FUNCTION_BLOCK FB_MotionAxisNCOld IMPLEMENTS I_MotionAxisOld
VAR
    iHome : I_Home;
    iHalt : I_Halt;
    iPower : I_Power;
    iReset : I_Reset;
    iMoveAbsolute : I_MoveAbsolute;
    iReadParameter : I_ReadParameter;
    iWriteParameter  : I_WriteParameter;
    iParamSaveRestore: I_ParamSaveRestore;
    iEncoderScaling : I_EncoderScaling;
    iAxisStatus : I_AxisStatus;
    iBacklashCompensation : I_BacklashCompensation;
    bError: BOOL;
    nErrorID: UDINT;
    sMessage : T_MAXSTRING;
    rtAbortDone : R_TRIG;

END_VAR

(*
    Error from NC functions
    The error will be sent to EPICS interface based on predifined
    priority: axis, power, backlash, absoluteMove, etc...
*)
IF THIS^.iPower.Error AND THIS^.iPower.PowerIsEnabled THEN
    bError:=THIS^.iPower.Error;
    nErrorId:=THIS^.iPower.ErrorID;
    sMessage := THIS^.iPower.Message;
ELSIF THIS^.iHalt.Error AND THIS^.iHalt.Active THEN
    bError:=THIS^.iHalt.Error;
    nErrorId:=THIS^.iHalt.ErrorID;
    sMessage := THIS^.iHalt.Message;
ELSIF THIS^.iReset.Error AND THIS^.iReset.Active THEN
    bError:=THIS^.iReset.Error;
    nErrorId:=THIS^.iReset.ErrorID;
    sMessage := THIS^.iReset.Message;
ELSIF THIS^.iBacklashCompensation.Error THEN
    bError:=THIS^.iBacklashCompensation.Error;
    nErrorId:=THIS^.iBacklashCompensation.ErrorID;
    sMessage := THIS^.iBacklashCompensation.Message;
ELSIF THIS^.iMoveAbsolute.Error THEN
    bError:=THIS^.iMoveAbsolute.Error;
    nErrorId:=THIS^.iMoveAbsolute.ErrorID;
    sMessage := THIS^.iMoveAbsolute.Message;
ELSIF THIS^.iHome.Error (*Homing error*) THEN
    bError:=THIS^.iHome.Error;
    nErrorId:=THIS^.iHome.ErrorID;
    sMessage := THIS^.iHome.Message;
ELSIF THIS^.iAxisStatus.Error  THEN
    bError:=THIS^.iAxisStatus.Error;
    nErrorId:=THIS^.iAxisStatus.ErrorID;
    sMessage := THIS^.iAxisStatus.Message;
ELSIF THIS^.iReadParameter.Error THEN
    bError := THIS^.iReadParameter.Error;
    nErrorId := THIS^.iReadParameter.ErrorID;
    sMessage := THIS^.iReadParameter.Message;
ELSIF THIS^.iWriteParameter.Error THEN
    bError := THIS^.iWriteParameter.Error;
    nErrorId := THIS^.iWriteParameter.ErrorID;
    sMessage := THIS^.iWriteParameter.Message;
ELSIF THIS^.iParamSaveRestore.Error THEN
    bError := THIS^.iParamSaveRestore.Error;
    nErrorId := THIS^.iParamSaveRestore.ErrorID;
    sMessage := THIS^.iParamSaveRestore.Message;
ELSE
    bError:=FALSE;
    nErrorId:=0;
    sMessage := '';
END_IF;

PROPERTY AbortDone : BOOL
GET
AbortDone := THIS^.iHalt.Done OR THIS^.iReset.Done;
END_GET
END_PROPERTY

PROPERTY Aborted : BOOL
GET
ABorted := THIS^.iMoveAbsolute.Aborted;
END_GET
END_PROPERTY

METHOD AxisEnabled : BOOL
VAR_INPUT
END_VAR
AxisEnabled:=THIS^.iAxisStatus.AxisEnabled();
END_METHOD

PROPERTY AxisReadParamsInit : BOOL
GET
AxisReadParamsInit := THIS^.iReadParameter.AxisReadParamsInit;
END_GET
END_PROPERTY

PROPERTY AxisState : MC_AxisStates
GET
AxisState := THIS^.iAxisStatus.AxisState;
END_GET
END_PROPERTY

(*
    Handle positive/negative backlash compensation
    User needs to set the direction of backlash from the sign of the compensation value
    Backlash compensation is disabled during referencing (homing).
    When direction is positive/negative, further movement in the negative/positive direction not compensated
    further movement in the negative/positive direction will be compensated
*)
METHOD BacklashCompensation
VAR_INPUT
	Enable : BOOL;
    BacklashComp: LREAL := 0.0;
    RampVelo : LREAL := 0.0;
END_VAR
THIS^.iBacklashCompensation.BacklashCompensation(	Enable:=Enable,
													RampVelo:=RampVelo
                                                );
END_METHOD

PROPERTY BacklashCompensationStatus : BOOL
GET
BacklashCompensationStatus := THIS^.iBacklashCompensation.Status;
END_GET
END_PROPERTY

PROPERTY Busy : BOOL
GET
Busy := THIS^.iHome.Busy OR THIS^.iMoveAbsolute.Busy;
END_GET
END_PROPERTY

METHOD PUBLIC CallAfterInit
VAR_INPUT
    iHome : I_Home;
    iHalt : I_Halt;
    iPower : I_Power;
    iReset : I_Reset;
    iMoveAbsolute : I_MoveAbsolute;
    iReadParameter : I_ReadParameter;
    iWriteParameter  : I_WriteParameter;
    iParamSaveRestore: I_ParamSaveRestore;
    iEncoderScaling : I_EncoderScaling;
    iAxisStatus : I_AxisStatus;
    iBacklashCompensation : I_BacklashCompensation;
END_VAR
THIS^.iHome := iHome;
THIS^.iHalt := iHalt;
THIS^.iPower := iPower;
THIS^.iReset := iReset;
THIS^.iMoveAbsolute := iMoveAbsolute;
THIS^.iReadParameter := iReadParameter ;
THIS^.iWriteParameter  := iWriteParameter;
THIS^.iParamSaveRestore:= iParamSaveRestore;
THIS^.iEncoderScaling := iEncoderScaling;
THIS^.iAxisStatus := iAxisStatus;
THIS^.iBacklashCompensation  := iBacklashCompensation ;
END_METHOD

PROPERTY Done : BOOL
GET
Done := THIS^.iHome.Done OR THIS^.iMoveAbsolute.Done;
END_GET
END_PROPERTY

METHOD DriveCommands
VAR_INPUT
    HomeCmd	: BOOL;
    NewMoveReq	: BOOL;
    EnableMode	: E_StageEnableMode;
END_VAR
END_METHOD

PROPERTY Error : BOOL
GET
Error := bError;
END_GET
END_PROPERTY

METHOD ErrorHandling
(*
    Error from functions and Nc
    The error will send to EPICS interface based on predifined
    priority: axis, power, backlash, absoluteMove, etc...
*)
IF THIS^.iAxisStatus.Error  THEN
    bError:=THIS^.iAxisStatus.Error;
    nErrorId:=THIS^.iAxisStatus.ErrorID;
    sMessage := THIS^.iAxisStatus.Message;
ELSIF THIS^.iPower.Error AND THIS^.iPower.PowerIsEnabled THEN
    bError:=THIS^.iPower.Error;
    nErrorId:=THIS^.iPower.ErrorID;
    sMessage := THIS^.iPower.Message;
ELSIF THIS^.iBacklashCompensation.Error THEN
    bError:=THIS^.iBacklashCompensation.Error;
    nErrorId:=THIS^.iBacklashCompensation.ErrorID;
    sMessage := THIS^.iBacklashCompensation.Message;
ELSIF THIS^.iMoveAbsolute.Error THEN
    bError:=THIS^.iMoveAbsolute.Error;
    nErrorId:=THIS^.iMoveAbsolute.ErrorID;
    sMessage := THIS^.iMoveAbsolute.Message;
ELSIF THIS^.iHome.Error (*Homing error*) THEN
    bError:=THIS^.iHome.Error;
    nErrorId:=THIS^.iHome.ErrorID;
    sMessage := THIS^.iHome.Message;
ELSIF THIS^.iHalt.Error AND THIS^.iHalt.Active THEN
    bError:=THIS^.iHalt.Error;
    nErrorId:=THIS^.iHalt.ErrorID;
    sMessage := THIS^.iHalt.Message;
ELSIF THIS^.iReset.Error  THEN
    bError:=THIS^.iReset.Error;
    nErrorId:=THIS^.iReset.ErrorID;
    sMessage := THIS^.iReset.Message;
ELSIF THIS^.iReadParameter.Error THEN
    bError := THIS^.iReadParameter.Error;
    nErrorId := THIS^.iReadParameter.ErrorID;
    sMessage := THIS^.iReadParameter.Message;
ELSIF THIS^.iWriteParameter.Error THEN
    bError := THIS^.iWriteParameter.Error;
    nErrorId := THIS^.iWriteParameter.ErrorID;
    sMessage := THIS^.iWriteParameter.Message;
ELSIF THIS^.iParamSaveRestore.Error THEN
    bError := THIS^.iParamSaveRestore.Error;
    nErrorId := THIS^.iParamSaveRestore.ErrorID;
    sMessage := THIS^.iParamSaveRestore.Message;
ELSE
    bError:=FALSE;
    nErrorId:=0;
    sMessage := '';
END_IF;
END_METHOD

PROPERTY ErrorID : UDINT
GET
ErrorID := THIS^.nErrorID;
END_GET
END_PROPERTY

//FB_Init is always available implicitly and it is used primarily for initialization.
//The return value is not evaluated. For a specific influence, you can also declare the
//methods explicitly and provide additional code there with the standard initialization
//code. You can evaluate the return value.
METHOD FB_Init: BOOL
VAR_INPUT
    bInitRetains: BOOL; // TRUE: the retain variables are initialized (reset warm / reset cold)
    bInCopyCode: BOOL;  // TRUE: the instance will be copied to the copy code afterward (online change)

    iHome : I_Home;
    iHalt : I_Halt;
    iPower : I_Power;
    iReset : I_Reset;
    iMoveAbsolute : I_MoveAbsolute;
    iReadParameter : I_ReadParameter;
    iWriteParameter  : I_WriteParameter;
    iParamSaveRestore: I_ParamSaveRestore;
    iEncoderScaling : I_EncoderScaling;
    iAxisStatus : I_AxisStatus;
    iBacklashCompensation : I_BacklashCompensation;
END_VAR
THIS^.iHome := iHome;
THIS^.iHalt := iHalt;
THIS^.iPower := iPower;
THIS^.iReset := iReset;
THIS^.iMoveAbsolute := iMoveAbsolute;
THIS^.iReadParameter := iReadParameter ;
THIS^.iWriteParameter  := iWriteParameter;
THIS^.iParamSaveRestore:= iParamSaveRestore;
THIS^.iEncoderScaling := iEncoderScaling;
THIS^.iAxisStatus := iAxisStatus;
THIS^.iBacklashCompensation  := iBacklashCompensation ;
END_METHOD

METHOD Halt
VAR_INPUT
    Deceleration	: LREAL := 0;
    Jerk	: LREAL := 0;
    BufferMode	: MC_BufferMode := MC_BufferMode.MC_Aborting;
END_VAR
THIS^.iHalt.Halt( 	Deceleration:=Deceleration,
                    Jerk:=Jerk ,
                    BufferMode:=BufferMode );
END_METHOD

PROPERTY HaltActive : BOOL
GET
HaltActive := THIS^.iHalt.Active;
END_GET
END_PROPERTY

PROPERTY HaltBusy : BOOL
GET
HaltBusy := THIS^.iHalt.Busy;
END_GET
END_PROPERTY

PROPERTY HaltDone : BOOL
GET
HaltDone := THIS^.iHalt.Done;
END_GET
END_PROPERTY

METHOD Home
VAR_INPUT
    Position        : LREAL         := DEFAULT_HOME_POSITION;
    BufferMode      : MC_BufferMode;
END_VAR
//
THIS^.iHome.Home(Position:=0.0,BufferMode:=MC_BufferMode.MC_Aborting);
END_METHOD

PROPERTY HomeBusy : BOOL
GET
HomeBusy := THIS^.iHome.Busy;
END_GET
END_PROPERTY

PROPERTY HomeDone : BOOL
GET
HomeDone := THIS^.iHome.Done;
END_GET
END_PROPERTY

PROPERTY HomeMode : E_EpicsHomeCmd
GET
HomeMode := THIS^.iHome.Mode;
END_GET
END_PROPERTY

PROPERTY InTargetPosition : BOOL
GET
InTargetPosition := THIS^.iAxisStatus.InTargetPosition;
END_GET
END_PROPERTY

PROPERTY MeasuredAcceleration : LREAL
GET
MeasuredAcceleration := THIS^.iAxisStatus.MeasuredAcceleration;
END_GET
END_PROPERTY

PROPERTY MeasuredCompensation : LREAL
GET
MeasuredCompensation := THIS^.iBacklashCompensation.CurrentBacklash;
END_GET
END_PROPERTY

PROPERTY MeasuredPosition : LREAL
GET
MeasuredPosition := THIS^.iAxisStatus.MeasuredPosition;
END_GET
END_PROPERTY

PROPERTY MeasuredPositionDiff : LREAL
GET
MeasuredPositionDiff := THIS^.iAxisStatus.MeasuredPositionDiff;
END_GET
END_PROPERTY

PROPERTY MeasuredVelocity : LREAL
GET
MeasuredVelocity := THIS^.iAxisStatus.MeasuredVelocity;
END_GET
END_PROPERTY

PROPERTY Message : T_MaxString
GET
Message :=sMessage;
END_GET
END_PROPERTY

METHOD MoveAbsolute
VAR_INPUT
    Position	: LREAL;
    Velocity	: LREAL;
    Acceleration	: LREAL := 0.0;
    Deceleration	: LREAL := 0.0;
    Jerk	: LREAL := 0.0;
    BufferMode	: MC_BufferMode := MC_BufferMode.MC_Aborting;
END_VAR
THIS^.iMoveAbsolute.MoveAbsolute( 	Position:=Position,
                                       Velocity := Velocity,
                                    Acceleration := Acceleration,
                                    Deceleration := Deceleration,
                                    Jerk := Jerk,
                                    BufferMode := BufferMode);
END_METHOD

PROPERTY MoveAbsoluteAborted : BOOL
GET
MoveAbsoluteAborted := THIS^.iMoveAbsolute.Aborted;
END_GET
END_PROPERTY

PROPERTY MoveAbsoluteActive : BOOL
GET
 MoveAbsoluteActive := THIS^.iMoveAbsolute.Active;
END_GET
END_PROPERTY

PROPERTY MoveAbsoluteBusy : BOOL
GET
MoveAbsoluteBusy := THIS^.iMoveAbsolute.Busy;
END_GET
END_PROPERTY

PROPERTY MoveAbsoluteDone : BOOL
GET
MoveAbsoluteDone := THIS^.iMoveAbsolute.Done;
END_GET
END_PROPERTY

PROPERTY NegativeMotionIsEnabled : BOOL
GET
 NegativeMotionIsEnabled := THIS^.iAxisStatus.NegativeMotionIsEnabled;
END_GET
END_PROPERTY

PROPERTY PositiveMotionIsEnabled : BOOL
GET
PositiveMotionIsEnabled := THIS^.iAxisStatus.PositiveMotionIsEnabled;
END_GET
END_PROPERTY

METHOD Power
VAR_INPUT
    Enable	: BOOL;
    Enable_Positive	: BOOL;
    Enable_Negative	: BOOL;
    Override	: LREAL := 100.0;
    BufferMode	: MC_BufferMode := MC_BufferMode.MC_Aborting;
END_VAR
THIS^.iPower.Power(	Enable:=Enable,
                    Enable_Positive:= Enable_Positive,
                    Enable_Negative:=Enable_Negative,
                    Override:=Override,
                    BufferMode:=BufferMode
                );
END_METHOD

PROPERTY PowerActive : BOOL
GET
PowerActive := THIS^.iPower.Active;
END_GET
END_PROPERTY

(*This is overriden by this object internal acess to the interlock instance
  this is intended to pass power enable flags via the fbMotionDrive
*)
METHOD PowerEnables
VAR_INPUT
    Enable	: BOOL;
    Enable_Positive	: BOOL;
    Enable_Negative	: BOOL;
END_VAR
THIS^.iPower.Power(	Enable:=Enable,
                    Enable_Positive:= Enable_Positive,
                    Enable_Negative:=Enable_Negative,
                    Override:=100.0,
                    BufferMode:=MC_BufferMode.MC_Aborting
                );
END_METHOD

PROPERTY PowerIsEnabled : BOOL
GET
END_GET
END_PROPERTY

PROPERTY PowerOverride : LREAL
GET
PowerOverride := THIS^.iPower.Override;
END_GET
END_PROPERTY

METHOD ReadAxisParams
VAR_INPUT
    Enable	: BOOL;
    RefreshDelay	: TIME;
END_VAR
THIS^.iReadParameter.ReadParameters(Enable:=Enable, RefreshDelay:=RefreshDelay);
END_METHOD

METHOD Reset
VAR_INPUT
END_VAR
THIS^.iReset.Reset();
END_METHOD

PROPERTY ResetBusy : BOOL
GET
ResetBusy := THIS^.iReset.Busy;
END_GET
END_PROPERTY

PROPERTY ResetDone : BOOL
GET
ResetDone := THIS^.iReset.Done;
END_GET
END_PROPERTY

PROPERTY RestoreDone : BOOL
GET
RestoreDone := THIS^.iParamSaveRestore.Done;
END_GET
END_PROPERTY

METHOD SaveAxisParams
VAR_INPUT
    Enable	: BOOL;
END_VAR
THIS^.iParamSaveRestore.SaveAxisParams(Enable:=Enable);
END_METHOD

PROPERTY SavedPosition : LREAL
GET
SavedPosition := THIS^.iParamSaveRestore.SavedPosition;
END_GET
END_PROPERTY

PROPERTY ScaledEncoderCount : UDINT
GET
ScaledEncoderCount := THIS^.iEncoderScaling.EncoderCount;
END_GET
END_PROPERTY

PROPERTY StandStill : BOOL
GET
StandStill := THIS^.iAxisStatus.StandStill;
END_GET
END_PROPERTY

(*
    Check all post condition before updating bCommandedMoveAbsolute
    The implmentatation will depend on the axis type
    DS402 NC/Direct axis : Implementation need to check that the drive is in the correct mode before initaiting the move then set bCommandedMoveAbsolute
    MP NC axis : will immediately write to bCommandedMoveAbsolute
*)
METHOD StartMove
VAR_INPUT
    MoveMode	: E_EpicsMotorCmd;
    CmdExecute	: BOOL;
END_VAR
END_METHOD

PROPERTY Stopped : BOOL
GET
Stopped := THIS^.iAxisStatus.Stopped;
END_GET
END_PROPERTY

END_FUNCTION_BLOCK

(* stored: Version 1.1.0.1
   POU FB_MotionAxisNCOld: Id {60e4ea75-36ff-4a14-b24a-51c7f7d1032f}, SpecialFunc None
   Property AbortDone: Id {1ab55f64-4d04-46ed-aa32-9a609a746501}
   Get Get: Id {5856cfc4-242e-4784-a316-d8c63bfdbc71}
   Property Aborted: Id {d0075b82-3e9e-46e5-acdf-4cebd8ebf67a}
   Get Get: Id {cf614298-ddff-4307-a171-563e96eb3c02}
   Method AxisEnabled: Id {e5e0c9e8-b45f-482d-9ef1-83edfb55d132}
   Property AxisReadParamsInit: Id {b8e5c5bb-b0b6-40eb-b5b6-dd5fb35ee51c}
   Get Get: Id {d8cc725d-08d5-44c2-b484-3f51796096a7}
   Property AxisState: Id {87002db8-c394-4716-a110-b766e1595838}
   Get Get: Id {c9f13994-021a-4c4e-998b-d440612ebd2e}
   Method BacklashCompensation: Id {1a08d8d8-a256-4b1e-88aa-d08b0121e4ae}
   Property BacklashCompensationStatus: Id {dbd09ba7-4925-432d-bcb3-61c45f839987}
   Get Get: Id {71a49803-cca5-4aae-a146-59674387d30e}
   Property Busy: Id {5e27d325-7e15-4c88-bfdb-3053f10f134b}
   Get Get: Id {55698422-4413-414b-bc0b-380708069192}
   Method CallAfterInit: Id {8a27238f-4890-4bb4-988b-8be7a7ea7777}
   Property Done: Id {e427a588-061f-4aa9-9222-7199e3e5682b}
   Get Get: Id {cef9feec-13b3-4b4a-8dc0-58a5b1ae0be4}
   Method DriveCommands: Id {da88f9ea-fae8-44f3-b945-ea433a793977}
   Property Error: Id {286c0d3a-410f-4676-aa62-a7393d4ea0e8}
   Get Get: Id {c8975688-24e7-4943-9f45-ac20d0000b11}
   Method ErrorHandling: Id {53078c0c-dd97-4634-ac7e-84052b41e871}
   Property ErrorID: Id {441bdd14-dc2f-4cc6-a8f8-fb710cc88bdf}
   Get Get: Id {100018d6-8d87-4c10-bcf7-592d27d6dad2}
   Method FB_Init: Id {3a0215de-bf6a-4c80-80c1-3b20f275bf2c}
   Method Halt: Id {8e589b74-150e-4146-8760-2ce7cd4c1a23}
   Property HaltActive: Id {77a509ea-ee54-4156-af92-101454fd556e}
   Get Get: Id {85b33736-4f99-4171-8039-29c3520477c2}
   Property HaltBusy: Id {cc24e04d-0fc3-4196-81f0-e034809ef886}
   Get Get: Id {0efdc27c-ea47-4a54-b0d5-ec69a2d31e31}
   Property HaltDone: Id {ebc24e4e-c40b-40fd-911f-a0d25bac9be2}
   Get Get: Id {35f34a04-8657-4c75-9f25-61a649e1024e}
   Method Home: Id {8a366a57-02cc-4b8d-a460-471eb54cdc9a}
   Property HomeBusy: Id {29ae59ac-7893-45dc-a7ff-d7afbb9a8eee}
   Get Get: Id {b1491b9a-862e-40d4-9b40-7b98da30786c}
   Property HomeDone: Id {a6cbb623-225a-4bca-bac2-d1b07cb33440}
   Get Get: Id {fa6132c9-1d9e-4aea-a5cf-9b2eba6f350e}
   Property HomeMode: Id {a6c014b5-da15-4ecb-b556-eeafc1302ddb}
   Get Get: Id {f2d86508-8281-4f5f-b43f-8f5e82346614}
   Property InTargetPosition: Id {c6f2b7e3-9865-497d-bb4f-27e1a950a6e2}
   Get Get: Id {7c6683fa-a37e-4085-91b2-78cfcff08531}
   Property MeasuredAcceleration: Id {7b279ce7-b390-4d74-b3ab-77fa9ef1e309}
   Get Get: Id {beb03da9-5519-4653-9d56-eba83a6b75e1}
   Property MeasuredCompensation: Id {92b62868-424e-4808-b20d-c6e6f7857102}
   Get Get: Id {dcff7040-9f93-42c7-bdab-ae8397de98c8}
   Property MeasuredPosition: Id {a15c9858-bafd-4376-84c9-f911bf0b147d}
   Get Get: Id {9d1af516-77e0-4dfa-8a39-31342ca2e8ea}
   Property MeasuredPositionDiff: Id {466798db-0628-4573-be15-482531f516a9}
   Get Get: Id {de73486e-ab47-4eaf-ae78-c6db5e2bb69f}
   Property MeasuredVelocity: Id {2668f40f-5052-4e32-b79b-05f0afca6340}
   Get Get: Id {83fc6d2e-1e55-4159-8d37-06c33fa4e8bc}
   Property Message: Id {26fc8d4c-3765-409d-99b9-88601f1c2c4a}
   Get Get: Id {667e5dee-2c71-4e47-9f4a-aaae83a2b01e}
   Method MoveAbsolute: Id {9a42793a-a8b6-4f1b-b7c4-807fd1695cd6}
   Property MoveAbsoluteAborted: Id {06d30932-17c7-4aba-a6bc-b4ba2774c3b9}
   Get Get: Id {d0c19c1f-74e8-4cca-8525-383dc0b1a139}
   Property MoveAbsoluteActive: Id {3a935e15-8cf5-4370-b49e-3b3eca7bbc95}
   Get Get: Id {1697a134-2850-4938-9960-40baeaa2a6e9}
   Property MoveAbsoluteBusy: Id {a9b2f63f-119d-43ce-9532-47639f98e2ff}
   Get Get: Id {0133b65b-8468-4a56-87a1-e37ae1ea3a84}
   Property MoveAbsoluteDone: Id {022dc82f-48a1-4f30-bc8e-5097d85d183f}
   Get Get: Id {a71688ae-b1b0-468d-9750-2bfd2cc9e180}
   Property NegativeMotionIsEnabled: Id {ab2e01ac-ef59-4eea-9e12-0071a5127d77}
   Get Get: Id {bc3a8001-ea55-4bfe-9303-f0182abdfcee}
   Property PositiveMotionIsEnabled: Id {216d3fb6-d257-47c0-b39c-b7449a269cdb}
   Get Get: Id {e3b922f5-7a0e-4dc5-a027-360a7ba73faf}
   Method Power: Id {2a90222a-cc04-4c30-9220-1a1e4e48ea37}
   Property PowerActive: Id {089621eb-ce6b-4c67-80c4-09fdf8f09b19}
   Get Get: Id {af8b06a3-efef-4599-96eb-64bd63e94e7c}
   Method PowerEnables: Id {f639508d-8ba3-4d48-9a88-1e3b26e91255}
   Property PowerIsEnabled: Id {3d454208-3930-4244-8f65-3c76dc064604}
   Get Get: Id {1db87986-5667-4e35-92e9-dde9f59a6a76}
   Property PowerOverride: Id {d996a2b4-35d6-4aa1-a9b5-8663398d418e}
   Get Get: Id {348e3b06-e009-4fce-acc9-9c0b4c2e7893}
   Method ReadAxisParams: Id {b4a17d98-327e-4fb3-91be-6ffbdb27eed3}
   Method Reset: Id {cd94c4b8-6191-42de-a670-30cee1e2d839}
   Property ResetBusy: Id {7f23536f-87d1-4a85-bf32-65e736b0c8b1}
   Get Get: Id {8667c29d-ea20-4889-8241-2482a1fcae47}
   Property ResetDone: Id {9780fa85-1310-4faa-95f1-4a520a1cc99c}
   Get Get: Id {05724d43-e9b9-44cb-987b-5fe07e4d39a2}
   Property RestoreDone: Id {6362c4f9-e739-4637-a9f5-2d26e4e0929f}
   Get Get: Id {92b0ecc0-faae-4950-bbdc-f0f30df9229b}
   Method SaveAxisParams: Id {b26155c4-7a52-4273-aab1-7b50f7613bd0}
   Property SavedPosition: Id {71101af8-1425-4601-8920-d5c3208896e2}
   Get Get: Id {046dc21b-acb5-46fb-8a70-b8ff3e1f2a94}
   Property ScaledEncoderCount: Id {b3991000-326d-4c42-a608-9c8991b7ccc5}
   Get Get: Id {c1b613be-7f1e-4301-a921-d5319255df56}
   Property StandStill: Id {4907e5fb-6983-4c1b-841e-8cbc707a3a49}
   Get Get: Id {101e5691-570a-4201-a10d-88a509f72d27}
   Method StartMove: Id {79bbc389-5cf8-4755-bad6-41240bbe8570}
   Property Stopped: Id {627971e5-8a4a-4a11-800c-3f489522ec58}
   Get Get: Id {bd33aa66-3078-4177-ac77-178f665dcc17} *)
